Fanuc KAREL source: kt00204.KL

-- PROVISIONAL review KL for V770-1; original PC SHA256 64963fb25b550d13a532ba6f0f2200c8dda7c727a2a9c22258a8afd40f20502d
-- Incomplete behavior may be omitted. Consult companion uncertainty JSON. Do not deploy.
PROGRAM KT00204
%NOLOCKGROUP
VAR
  I1 : INTEGER
  I2 : INTEGER
  OUT : INTEGER
BEGIN
  -- UNRESOLVED_PC offsets 5-16; opcodes 2E,23
  -- UNRESOLVED_PC offsets 21-32; opcodes 2E,23
  -- UNRESOLVED_PC offsets 37-48; opcodes 2E,23
  -- UNRESOLVED_PC offsets 53-64; opcodes 2E,23
  -- UNRESOLVED_PC offsets 69-88; opcodes 21,21,46,23
  -- UNRESOLVED_PC offsets 93-97; opcodes 7F
END KT00204
